FUNCTION_BLOCK T_ExternalControllersCollectionNotifyModeChangedSuccess EXTENDS T_UnitTestBase
VAR
  list : T_ExternalControllerCollection(10);
  newController, newController2 : T_ExternalControllerMock; 
  actual1, actual2 : BOOL;
END_VAR

// Arrange
list.AddController(newController);
list.AddController(newController2);

//Act
list.NotifyModeChanged(E_PMLUnitMode.ePMLUnitMode_Maintenance);

//Assert
actual1 := newController._newMode= E_PMLUnitMode.ePMLUnitMode_Maintenance;
actual2 := newController2._newMode = E_PMLUnitMode.ePMLUnitMode_Maintenance;

assertion.AssertEquals_BOOL(TRUE, actual1, 'newController._newState = Tc3_PackML_V2.E_PMLCommand.ePMLCommand_Complete');
assertion.AssertEquals_BOOL(TRUE, actual2, 'newController2._newState = Tc3_PackML_V2.E_PMLCommand.ePMLCommand_Complete');
TestFinished();

END_FUNCTION_BLOCK

(* stored: Version 1.1.0.1, ProductVersion 3.1.4024.12
   POU T_ExternalControllersCollectionNotifyModeChangedSuccess: Id {9aaeaa7d-3437-4364-9c4c-29673879c3af}, SpecialFunc None *)
